TYPE T_Map_Entry : ST_MAP_ENTRY; END_TYPE

(* stored: Version 1.1.0.1, ProductVersion 3.1.4024.4
   DUT T_Map_Entry: Id {a93d3904-e0b5-4d11-96e4-b0b8f7288243} *)
